PROGRAM PROG2
VAR
END_VAR

END_PROGRAM

(* stored: Version 1.1.0.1, ProductVersion 3.1.4024.5
   POU PROG2: Id {c1de8348-925f-4e8a-b45e-f1215222bb9d}, SpecialFunc None *)
